{attribute addProperty BoxType "EL4124-0000-1016"}
{attribute addProperty Id "AO_Output_ChannelAT %Q*ARRAY[0..3] OF AO_Output_Channel_F57FA4F96480WcStateAT %I*WcState_28A8677510.1250InfoDataAT %I*InfoData_BC63D37F80100"}
{attribute addProperty CRC "3820990709"}
{attribute addProperty SizeInBites "145"}
{attribute addProperty SizeInBytes "18.125"}
TYPE EL4124_FEE36ED0 :
STRUCT
	{attribute addProperty Name "AO_Output_Channel"}
	AO_Output_Channel : ARRAY[0..3] OF AO_Output_Channel_F57FA4F9;
	{attribute addProperty Name "WcState"}
	WcState : WcState_28A86775;
	{attribute addProperty Name "InfoData"}
	InfoData : InfoData_BC63D37F;
END_STRUCT
END_TYPE

(* stored: Version 1.2.0.0, ProductVersion 3.1.4024.9
   DUT EL4124_FEE36ED0: Id {a42d52f2-b1c8-4226-bd9e-7e309495ab1d} *)
